(* CODESYS project LD_TEST.xml

Project tree, tasks and I/O mapping:
  program LD_TEST [LD]
*)

// LD_TEST
PROGRAM LD_TEST
VAR
	Sensor1: BOOL;
	Sensor2: BOOL;
	sensor3: BOOL;
	PowerOn: BOOL;
	TON_0: TON;
	CTU_0: CTU;
	PowerOff: BOOL;
END_VAR

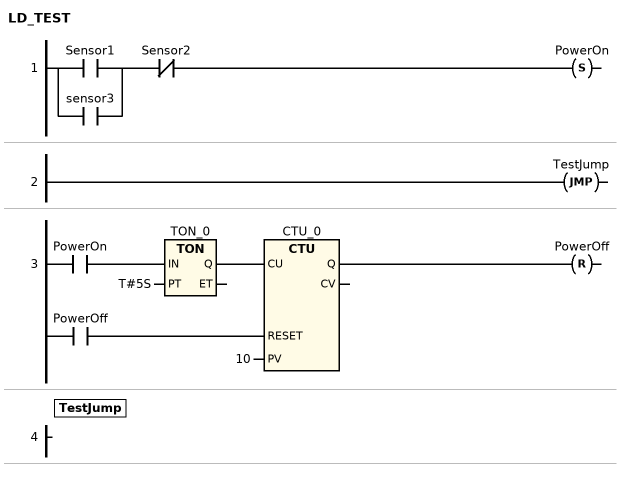
// NETWORK 1
PowerOn S= (Sensor1 OR sensor3) AND NOT Sensor2;

// NETWORK 2
JMP TestJump;

// NETWORK 3
TON_0(IN := PowerOn, PT := T#5S); // TON
CTU_0(CU := TON_0.Q, RESET := PowerOff, PV := 10); // CTU
PowerOff R= CTU_0.Q;

// NETWORK 4
TestJump: ;

END_PROGRAM
